// Passes cleanly, then hangs on the way out.

//

// The verdict must survive: a passing test whose cleanup hung still proved the

// code correct. The overrun is a framework error, not a test failure - but on a

// rig it may mean an axis left powered, so it must be loud.
FUNCTION_BLOCK HangingTeardownTest IMPLEMENTS I_Test, I_TestTeardown
VAR
	_BodyCalls	   : UDINT;
	_TeardownCalls : UDINT;
END_VAR

PROPERTY BodyCalls : UDINT
GET
BodyCalls := _BodyCalls;
END_GET
END_PROPERTY

METHOD Run : BOOL
VAR_INPUT
	Enable : BOOL;
	Test   : I_TestAssertions;
END_VAR
IF Enable THEN
	_BodyCalls := _BodyCalls + 1;
	Test.AssertTrue(TRUE, 'the body was fine');
END_IF

Run := TRUE;
END_METHOD

METHOD Teardown : BOOL
VAR_INPUT
	Enable : BOOL;
	Test   : I_TestAssertions;
END_VAR
IF Enable THEN
	_TeardownCalls := _TeardownCalls + 1;
END_IF

Teardown := FALSE;
END_METHOD

PROPERTY TeardownCalls : UDINT
GET
TeardownCalls := _TeardownCalls;
END_GET
END_PROPERTY

END_FUNCTION_BLOCK

(* stored: Version 1.1.0.1, ProductVersion 3.1.4026.18
   POU HangingTeardownTest: Id {c0f5c382-366d-4dc6-8b62-6a2c8ea627e7}, SpecialFunc None
   Folder I_Test: Id {26ca4b75-71ef-4df8-bbbc-9365d46f8316}
   Folder I_TestTeardown: Id {7e3dbd27-8147-439f-88e1-48d0c30c5bd6}
   Property BodyCalls: Id {784e5c86-6178-4e50-ba2a-3a900a62f392}
   Get Get: Id {18bf104e-ab74-4bdf-b206-2dabb67d4310}
   Method Run: Id {23b3dcfa-5008-400d-aaef-ec98e7cf3793}
   Method Teardown: Id {b81859d0-73dd-4d7d-8361-78e16f169fc1}
   Property TeardownCalls: Id {7fc8e838-f893-45a8-97d3-6e7945e97f39}
   Get Get: Id {17ad5b8a-ceaf-4d85-ad35-097de5ceaf37} *)
